// SIMATIC S7-200 project (STEP 7-Micro/WIN), CPU 224 CN REL 02.02

SYMBOL_TABLE 用户定义1
手自动选择            I0.0     // 系统手动/自动选择
搅拌机过载            I0.1     // 搅拌机过载
系统复位             I0.2     // 系统复位
放料阀手动            I0.3     // 放料阀手动
搅拌机手动            I0.4     // 搅拌机手动
取料阀手动            I0.5     // 取料阀手动
取料阀输出            Q0.0     // 取料阀输出
搅拌机输出            Q0.1     // 搅拌机输出
放料阀手输出           Q0.2     // 放料阀手输出
报警输出             Q0.3     // 报警输出
END_SYMBOL_TABLE

ORGANIZATION_BLOCK 主程序:OB1
TITLE=程序注释
BEGIN
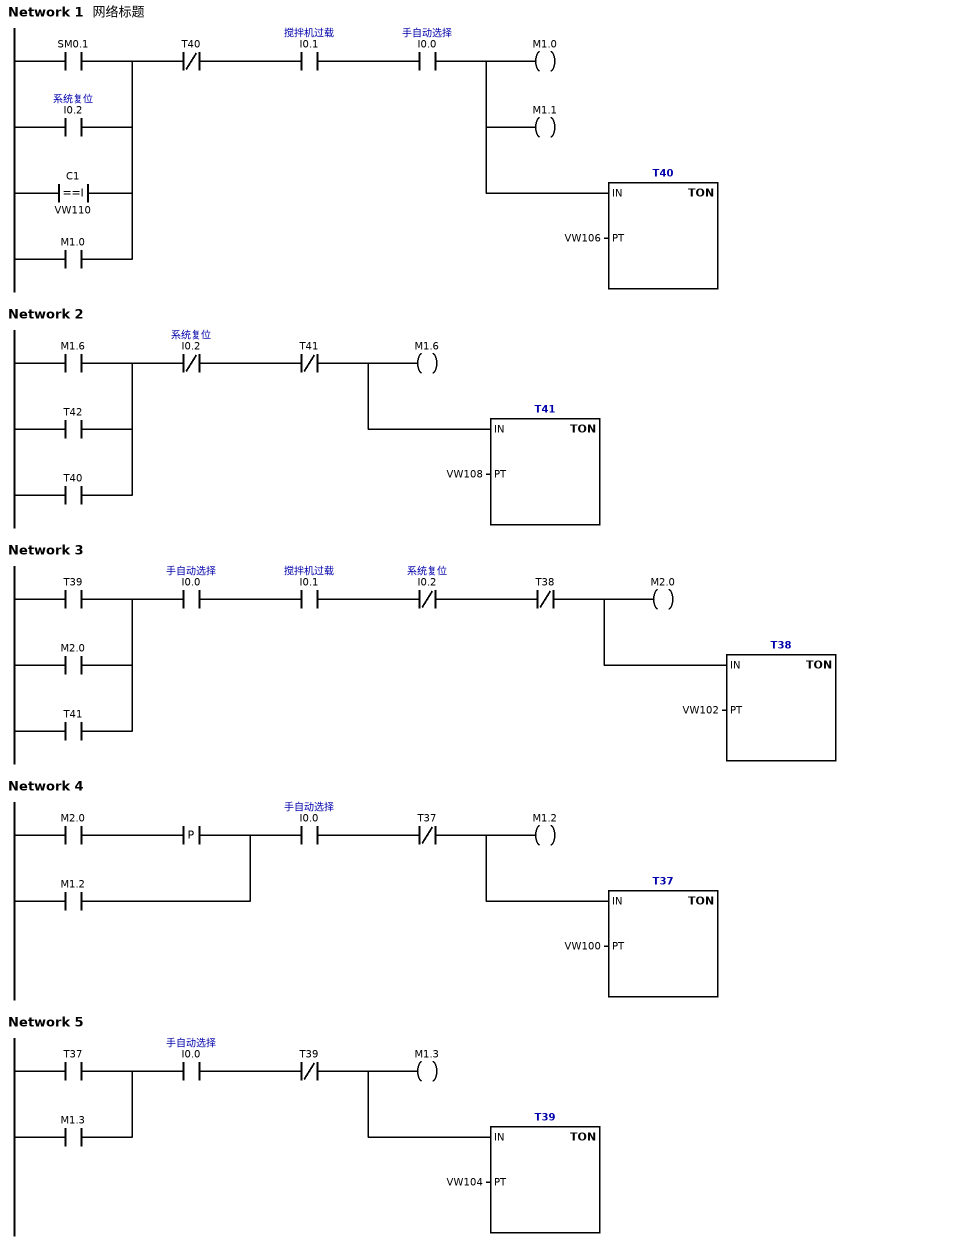
Network 1 // 网络标题
LD     SM0.1
O      系统复位:I0.2
OW=    C1, VW110
O      M1.0
AN     T40
A      搅拌机过载:I0.1
A      手自动选择:I0.0
=      M1.0
=      M1.1
TON    T40, VW106
Network 2
LD     M1.6
O      T42
O      T40
AN     系统复位:I0.2
AN     T41
=      M1.6
TON    T41, VW108
Network 3
LD     T39
O      M2.0
O      T41
A      手自动选择:I0.0
A      搅拌机过载:I0.1
AN     系统复位:I0.2
AN     T38
=      M2.0
TON    T38, VW102
Network 4
LD     M2.0
EU
O      M1.2
A      手自动选择:I0.0
AN     T37
=      M1.2
TON    T37, VW100
Network 5
LD     T37
O      M1.3
A      手自动选择:I0.0
AN     T39
=      M1.3
TON    T39, VW104
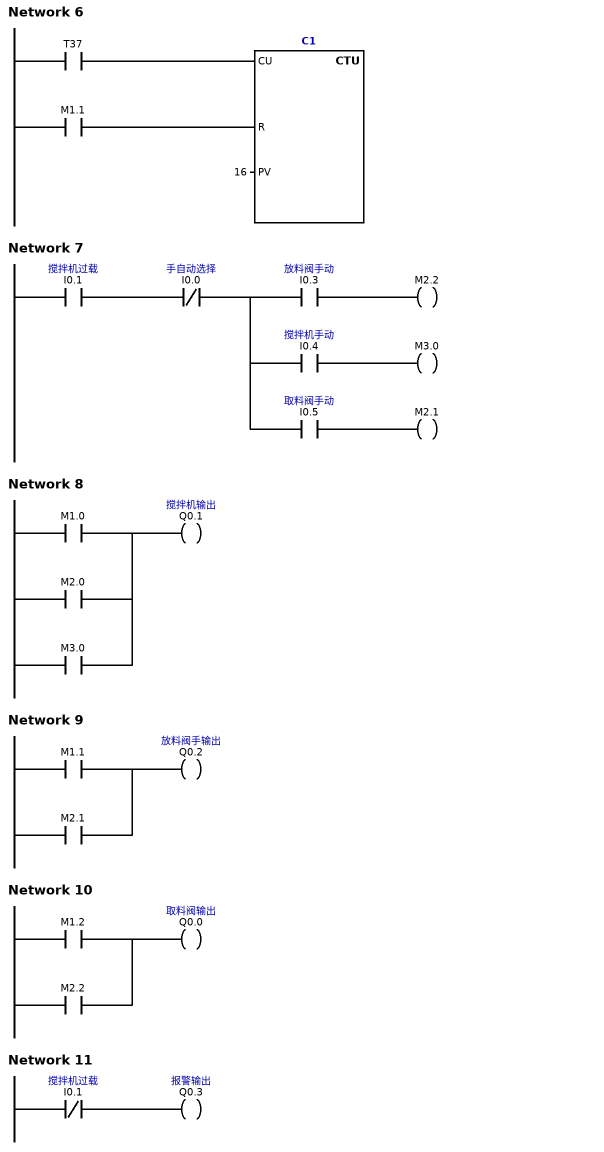
Network 6
// (network saved uncompiled; LAD cells follow)
// row 0: c0 -| |- T37  c1 --  c2 [CTU C1 CU:=power@row0, R:=power@row1, PV:=16]
// row 1: c0 -| |- M1.1  c1 --  c2 [box]
// row 2: c2 [box]
Network 7
LD     搅拌机过载:I0.1
AN     手自动选择:I0.0
LPS
A      放料阀手动:I0.3
=      M2.2
LRD
A      搅拌机手动:I0.4
=      M3.0
LPP
A      取料阀手动:I0.5
=      M2.1
Network 8
LD     M1.0
O      M2.0
O      M3.0
=      搅拌机输出:Q0.1
Network 9
LD     M1.1
O      M2.1
=      放料阀手输出:Q0.2
Network 10
LD     M1.2
O      M2.2
=      取料阀输出:Q0.0
Network 11
LDN    搅拌机过载:I0.1
=      报警输出:Q0.3
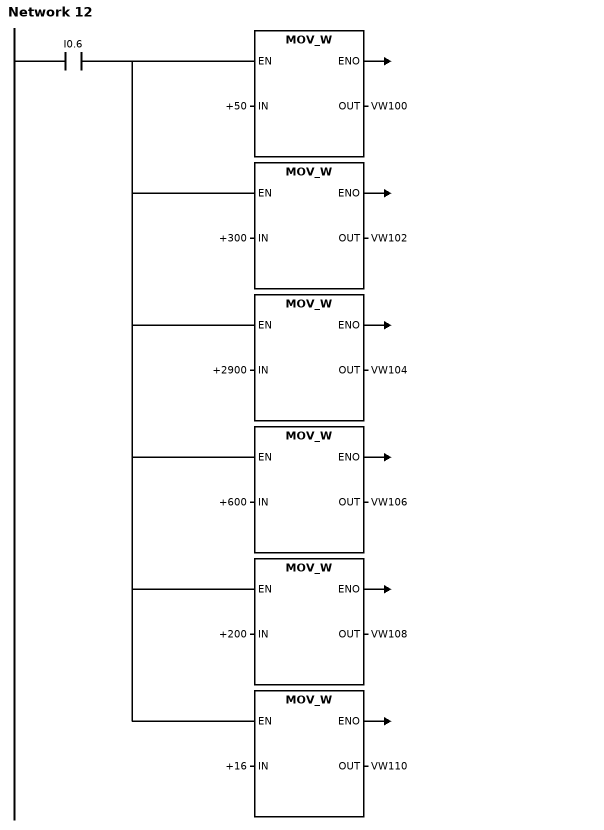
Network 12
LD     I0.6
MOVW   +50, VW100
MOVW   +300, VW102
MOVW   +2900, VW104
MOVW   +600, VW106
MOVW   +200, VW108
MOVW   +16, VW110
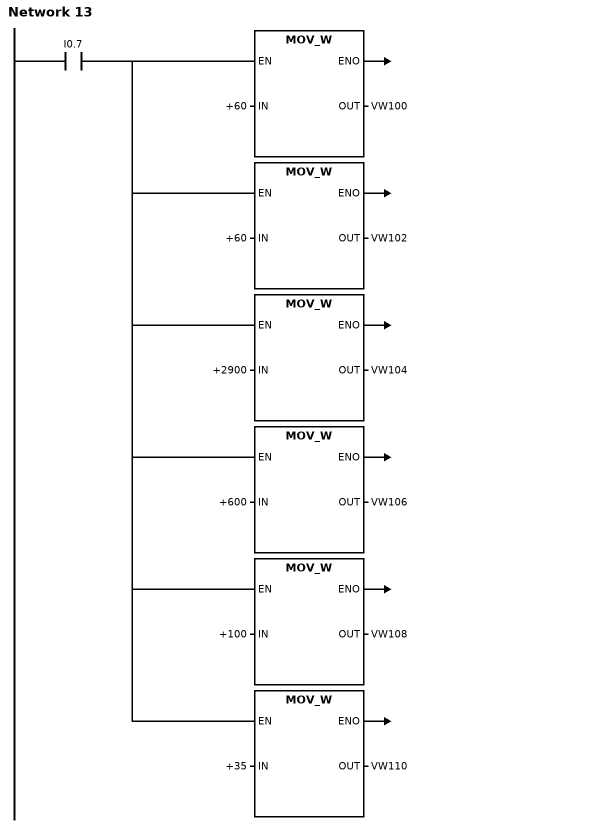
Network 13
LD     I0.7
MOVW   +60, VW100
MOVW   +60, VW102
MOVW   +2900, VW104
MOVW   +600, VW106
MOVW   +100, VW108
MOVW   +35, VW110
END_ORGANIZATION_BLOCK
